TYPE ST_DB_Config :
STRUCT

	bDBConfigured				: BOOL;
	sSQLName					: STRING;
	sDatabaseName				: STRING;
	stNetAddress				: ST_TCPIP_AddressPort;
	nLastDBID					: UDINT;

	bEnableOCVCheck							: BOOL;
	bEnableOACCheck							: BOOL;
	bEnableCACCheck							: BOOL;

END_STRUCT
END_TYPE

(* stored: Version 1.1.0.1
   DUT ST_DB_Config: Id {eaad5bcc-92b6-4ae4-a6c7-b1c70f5210a1} *)
